{attribute 'conditionalshow'}
FUNCTION_BLOCK FB_CV_INT_TO_WORD
VAR_INPUT
	{attribute 'hide'}
	iInputValue					: INT;								//Input value that is converted into the output value							
END_VAR
VAR_OUTPUT
	{attribute 'hide'}
	wOutputValue				: WORD;								//Converted output value
END_VAR
VAR
END_VAR

//Creator : Kai Ebensperger
//Company : Lynus AG
//Date : 28.04.2021
//Version : 1.0.0.0

//With this functionblock its possible to convert a certain Datatyp in a other Datatype
//INT TO WORD
//Created for the Edge Device Lib over Modbus TCP
//Modbus TCP is WORD oriented

wOutputValue := INT_TO_WORD(iInputValue);

END_FUNCTION_BLOCK

(* stored: Version 1.1.0.1, ProductVersion 3.1.4024.9
   POU FB_CV_INT_TO_WORD: Id {32cdf57d-dde4-448f-bf15-8c499b97e8a8}, SpecialFunc None *)
